KUKA KRL data list: bto.dat

&ACCESS RVP
&REL 2
&PARAM TEMPLATE = C:\KRC\Roboter\Template\vorgabe
&PARAM EDITMASK = *
DEFDAT BTO
;FOLD EXTERNAL DECLARATIONS;%{PE}%V3.2.0,%MKUKATPBASIS,%CEXT,%VCOMMON,%P
;FOLD BAS EXT;%{PE}%V3.2.0,%MKUKATPBASIS,%CEXT,%VEXT,%P
EXT  BAS (BAS_COMMAND  :IN,REAL  :IN )
DECL INT SUCCESS
;ENDFOLD
;FOLD A10 EXT;%{E}%V3.2.0,%MKUKATPARC,%CEXT,%VEXT,%P
EXT  A10 (A_CMD_T  :IN,A_STRT_T  :IN,A_WELD_T  :IN,A_END_T  :IN,INT  :IN )
;ENDFOLD
;FOLD A20 EXT;%{E}%V3.2.0,%MKUKATPA20,%CEXT,%VEXT,%P
EXT  A20 (INT  :IN,WELD_ST  :IN,WELD_FI  :IN,INT  :IN )
;ENDFOLD
;FOLD GRIPPER EXT;%{E}%V3.2.0,%MKUKATPGRIPPER,%CEXT,%VEXT,%P
EXT  H50 (INT  :IN,INT  :IN,INT  :IN,GRP_TYP  :IN )
;ENDFOLD
;FOLD SPOT EXT;%{E}%V3.2.0,%MKUKATPSPOT,%CEXT,%VEXT,%P
EXT  USERSPOT (S_COMMAND  :IN,SPOT_TYPE  :IN )
;ENDFOLD
;FOLD TOUCHSENSE EXT;%{E}%V3.2.0,%MKUKATPTS,%CEXT,%VEXT,%P
EXT  H70 (INT  :IN,SRCH_TYP_2  :OUT,E6POS  :IN,SRCH_TYP_3  :IN,SRCH_TYP_2  :IN,SRCH_TYP_2  :IN,SRCH_TYP_2  :IN,SRCH_TYP_2  :IN,SRCH_TYP_2  :IN,INT  :IN )
;ENDFOLD
;FOLD USER EXT;%{E}%V3.2.0,%MKUKATPUSER,%CEXT,%VEXT,%P
;Make here your modifications
;ENDFOLD
;ENDFOLD

DECL BASIS_SUGG_T LAST_BASIS={POINT1[] "Frente_de_cnc           ",POINT2[] "Frente_de_cnc           ",CP_PARAMS[] "CPDAT1                  ",PTP_PARAMS[] "PDAT1                   ",CONT[] "C_PTP                   ",CP_VEL[] "0.3                     ",PTP_VEL[] "10                      "}
DECL E6POS XFRENTECINTA={x 586.713501,y 475.164886,z 2277.23389,a 88.4521027,b -44.9880409,c -179.531097,s 2,t 43,e1 0.0,e2 0.0,e3 0.0,e4 0.0,e5 0.0,e6 0.0}
DECL FDAT FFrenteCinta={TOOL_NO 0,BASE_NO 0,IPO_FRAME #BASE}
DECL PDAT PPDAT1={VEL 100.0,ACC 100.0,APO_DIST 100.0}
DECL FDAT FFrenteCNC={TOOL_NO 0,BASE_NO 0,IPO_FRAME #BASE}
DECL E6POS XDEJARPINZA2CINTA={x 1620.00403,y -0.00337643898,z 1909.99402,a -110.582497,b 89.9985199,c -110.582397,s 2,t 2,e1 0.0,e2 0.0,e3 0.0,e4 0.0,e5 0.0,e6 0.0}
DECL FDAT FDejarPinza2Cinta={TOOL_NO 2,BASE_NO 0,IPO_FRAME #BASE}
DECL PDAT PPDAT2={VEL 100.0,ACC 100.0,APO_DIST 100.0}
DECL E6POS XDEJARPINZA1CINTA={x -822.804382,y 1453.90796,z 1167.45105,a 3.40687394,b 43.3361893,c -176.740799,s 2,t 35,e1 0.0,e2 0.0,e3 0.0,e4 0.0,e5 0.0,e6 0.0}
DECL FDAT FDejarPinza1Cinta={TOOL_NO 1,BASE_NO 0,IPO_FRAME #BASE}
DECL PDAT PPDAT3={VEL 100.0,ACC 100.0,APO_DIST 100.0}
DECL E6POS XENT1_COGERCINTA={x 444.522186,y 912.39978,z 1228.745,a 87.1254272,b -7.41709614,c -179.732895,s 2,t 43,e1 0.0,e2 0.0,e3 0.0,e4 0.0,e5 0.0,e6 0.0}
DECL FDAT FEnt1_CogerCinta={TOOL_NO 1,BASE_NO 0,IPO_FRAME #BASE}
DECL PDAT PPDAT4={VEL 100.0,ACC 100.0,APO_DIST 100.0}
DECL E6POS XENT2_COGERCINTA={x 175.7229,y 1220.86304,z 1143.29395,a 91.0016403,b -16.5721092,c -179.742203,s 2,t 43,e1 0.0,e2 0.0,e3 0.0,e4 0.0,e5 0.0,e6 0.0}
DECL FDAT FEnt2_CogerCinta={TOOL_NO 1,BASE_NO 0,IPO_FRAME #BASE}
DECL PDAT PPDAT5={VEL 100.0,ACC 100.0,APO_DIST 100.0}
DECL E6POS XENT3COGERCINTA={x 174.258408,y 1264.94495,z 995.101624,a 91.0015488,b -16.5722103,c -179.742203,s 2,t 43,e1 0.0,e2 0.0,e3 0.0,e4 0.0,e5 0.0,e6 0.0}
DECL FDAT FEnt3CogerCinta={TOOL_NO 1,BASE_NO 0,IPO_FRAME #BASE}
DECL PDAT PPDAT6={VEL 100.0,ACC 100.0,APO_DIST 100.0}
DECL LDAT LCPDAT1={VEL 2.0,ACC 100.0,APO_DIST 100.0,APO_FAC 50.0}
DECL E6POS XCOGERCINTA={x 172.789902,y 1308.08704,z 849.818787,a 91.0006485,b -16.5677299,c -179.738998,s 2,t 43,e1 0.0,e2 0.0,e3 0.0,e4 0.0,e5 0.0,e6 0.0}
DECL FDAT FCogerCinta={TOOL_NO 1,BASE_NO 0,IPO_FRAME #BASE}
DECL LDAT LCPDAT2={VEL 2.0,ACC 100.0,APO_DIST 100.0,APO_FAC 50.0}
DECL E6POS XSAL1_COGERCINTA={x 174.258408,y 1264.94495,z 995.101624,a 91.0015488,b -16.5722103,c -179.742203,s 2,t 43,e1 0.0,e2 0.0,e3 0.0,e4 0.0,e5 0.0,e6 0.0}
DECL FDAT FSal1_CogerCinta={TOOL_NO 1,BASE_NO 0,IPO_FRAME #BASE}
DECL LDAT LCPDAT3={VEL 2.0,ACC 100.0,APO_DIST 100.0,APO_FAC 50.0}
DECL E6POS XSAL2_COGERCINTA={x 175.7229,y 1220.86304,z 1143.29395,a 91.0016403,b -16.5721092,c -179.742203,s 2,t 43,e1 0.0,e2 0.0,e3 0.0,e4 0.0,e5 0.0,e6 0.0}
DECL FDAT FSal2_CogerCinta={TOOL_NO 1,BASE_NO 0,IPO_FRAME #BASE}
DECL PDAT PPDAT7={VEL 100.0,ACC 100.0,APO_DIST 100.0}
DECL E6POS XENT1_COGERCNC={x 1664.62,y -787.04303,z 1556.33203,a 3.4404459,b -72.5609131,c 178.200897,s 2,t 42,e1 0.0,e2 0.0,e3 0.0,e4 0.0,e5 0.0,e6 0.0}
DECL FDAT FEnt1_CogerCNC={TOOL_NO 2,BASE_NO 0,IPO_FRAME #BASE}
DECL PDAT PPDAT8={VEL 100.0,ACC 100.0,APO_DIST 100.0}
DECL E6POS XENT2_COGERCNC={x 1791.36096,y -713.231323,z 1242.87,a 2.15886807,b -62.4185295,c 177.698502,s 2,t 42,e1 0.0,e2 0.0,e3 0.0,e4 0.0,e5 0.0,e6 0.0}
DECL FDAT FEnt2_CogerCNC={TOOL_NO 2,BASE_NO 0,IPO_FRAME #BASE}
DECL PDAT PPDAT9={VEL 100.0,ACC 100.0,APO_DIST 100.0}
DECL E6POS XENT3_COGERCNC={x 1968.31201,y -714.600403,z 1150.51599,a 2.13476205,b -62.4179115,c 177.698898,s 2,t 42,e1 0.0,e2 0.0,e3 0.0,e4 0.0,e5 0.0,e6 0.0}
DECL FDAT FEnt3_CogerCNC={TOOL_NO 2,BASE_NO 0,IPO_FRAME #BASE}
DECL LDAT LCPDAT4={VEL 2.0,ACC 100.0,APO_DIST 100.0,APO_FAC 50.0}
DECL E6POS XCOGERCNC={x 2122.44507,y -715.841675,z 1070.07898,a 2.13489294,b -62.4179802,c 177.6987,s 2,t 42,e1 0.0,e2 0.0,e3 0.0,e4 0.0,e5 0.0,e6 0.0}
DECL FDAT FCogerCNC={TOOL_NO 2,BASE_NO 0,IPO_FRAME #BASE}
DECL LDAT LCPDAT5={VEL 2.0,ACC 100.0,APO_DIST 100.0,APO_FAC 50.0}
DECL E6POS XSAL1_COGERCNC={x 2122.44702,y -750.182312,z 1070.07996,a 2.13447905,b -62.4182396,c 177.698898,s 2,t 42,e1 0.0,e2 0.0,e3 0.0,e4 0.0,e5 0.0,e6 0.0}
DECL FDAT FSal1_CogerCNC={TOOL_NO 2,BASE_NO 0,IPO_FRAME #BASE}
DECL LDAT LCPDAT6={VEL 2.0,ACC 100.0,APO_DIST 100.0,APO_FAC 50.0}
DECL E6POS XSAL2_COGERCNC={x 2303.74194,y -787.196472,z 1397.98206,a 2.13354492,b -62.4185104,c 177.699097,s 2,t 42,e1 0.0,e2 0.0,e3 0.0,e4 0.0,e5 0.0,e6 0.0}
DECL FDAT FSal2_CogerCNC={TOOL_NO 2,BASE_NO 0,IPO_FRAME #BASE}
DECL LDAT LCPDAT7={VEL 2.0,ACC 100.0,APO_DIST 100.0,APO_FAC 50.0}
DECL E6POS XENT1_DEJARCNC={x 2008.724,y -885.728271,z 1470.271,a 1.25756299,b -55.0479698,c -179.549301,s 2,t 42,e1 0.0,e2 0.0,e3 0.0,e4 0.0,e5 0.0,e6 0.0}
DECL FDAT FEnt1_DejarCNC={TOOL_NO 1,BASE_NO 0,IPO_FRAME #BASE}
DECL PDAT PPDAT10={VEL 100.0,ACC 100.0,APO_DIST 100.0}
DECL E6POS XENT2_DEJARCNC={x 2273.48389,y -808.585876,z 1205.05798,a 1.25766599,b -55.0479317,c -179.549606,s 2,t 42,e1 0.0,e2 0.0,e3 0.0,e4 0.0,e5 0.0,e6 0.0}
DECL FDAT FEnt2_DejarCNC={TOOL_NO 1,BASE_NO 0,IPO_FRAME #BASE}
DECL PDAT PPDAT11={VEL 100.0,ACC 100.0,APO_DIST 100.0}
DECL E6POS XENT3_DEJARCNC={x 2114.40503,y -752.901978,z 1057.99695,a 1.25682998,b -55.0801506,c -179.549698,s 2,t 42,e1 0.0,e2 0.0,e3 0.0,e4 0.0,e5 0.0,e6 0.0}
DECL FDAT FEnt3_DejarCNC={TOOL_NO 1,BASE_NO 0,IPO_FRAME #BASE}
DECL LDAT LCPDAT8={VEL 2.0,ACC 100.0,APO_DIST 100.0,APO_FAC 50.0}
DECL E6POS XDEJARCNC={x 2113.43701,y -718.692322,z 1058.151,a 1.25690103,b -55.0800896,c -179.556305,s 2,t 42,e1 0.0,e2 0.0,e3 0.0,e4 0.0,e5 0.0,e6 0.0}
DECL FDAT FDejarCNC={TOOL_NO 1,BASE_NO 0,IPO_FRAME #BASE}
DECL LDAT LCPDAT9={VEL 2.0,ACC 100.0,APO_DIST 100.0,APO_FAC 50.0}
DECL E6POS XSAL1_CNC={x 2037.91797,y -721.06012,z 1110.89697,a 1.25862098,b -55.0801697,c -179.557907,s 2,t 42,e1 0.0,e2 0.0,e3 0.0,e4 0.0,e5 0.0,e6 0.0}
DECL FDAT FSal1_CNC={TOOL_NO 1,BASE_NO 0,IPO_FRAME #BASE}
DECL LDAT LCPDAT10={VEL 2.0,ACC 100.0,APO_DIST 100.0,APO_FAC 50.0}
DECL E6POS XSAL2_CNC={x 1572.76794,y -714.070374,z 1503.53406,a 0.854870021,b -43.0494003,c -179.635498,s 2,t 42,e1 0.0,e2 0.0,e3 0.0,e4 0.0,e5 0.0,e6 0.0}
DECL FDAT FSal2_CNC={TOOL_NO 1,BASE_NO 0,IPO_FRAME #BASE}
DECL PDAT PPDAT12={VEL 100.0,ACC 100.0,APO_DIST 100.0}
DECL E6POS XSAL3_CNC={x 1229.31995,y -808.674805,z 1490.52698,a 2.84506607,b -24.9072895,c 179.859299,s 2,t 42,e1 0.0,e2 0.0,e3 0.0,e4 0.0,e5 0.0,e6 0.0}
DECL FDAT FSal3_CNC={TOOL_NO 1,BASE_NO 0,IPO_FRAME #BASE}
DECL PDAT PPDAT13={VEL 100.0,ACC 100.0,APO_DIST 100.0}
DECL PDAT PPDAT14={VEL 100.0,ACC 100.0,APO_DIST 100.0}
DECL E6POS XENT1_DEJARCINTA={x -732.870728,y 1158.88794,z 2270.01904,a 59.0703812,b -89.6684494,c -91.9009628,s 2,t 43,e1 0.0,e2 0.0,e3 0.0,e4 0.0,e5 0.0,e6 0.0}
DECL FDAT FEnt1_DejarCinta={TOOL_NO 2,BASE_NO 0,IPO_FRAME #BASE}
DECL PDAT PPDAT15={VEL 100.0,ACC 100.0,APO_DIST 100.0}
DECL E6POS XENT2_DEJARCINTA={x -1001.48102,y 1524.125,z 1379.88904,a -179.701401,b -42.7616196,c 178.789902,s 2,t 35,e1 0.0,e2 0.0,e3 0.0,e4 0.0,e5 0.0,e6 0.0}
DECL FDAT FEnt2_DejarCinta={TOOL_NO 2,BASE_NO 0,IPO_FRAME #BASE}
DECL PDAT PPDAT16={VEL 100.0,ACC 100.0,APO_DIST 100.0}
DECL E6POS XSAL1_DEJARCINTA={x -732.870728,y 1158.88794,z 2270.01904,a 59.0703812,b -89.6684494,c -91.9009628,s 2,t 43,e1 0.0,e2 0.0,e3 0.0,e4 0.0,e5 0.0,e6 0.0}
DECL FDAT FSal1_DejarCinta={TOOL_NO 2,BASE_NO 0,IPO_FRAME #BASE}
DECL PDAT PPDAT17={VEL 100.0,ACC 100.0,APO_DIST 100.0}
DECL GRP_SUGG_T LAST_GRP={NUMBER[] "2                       ",STATE[] "1                       ",PARAMS[] "GDAT7                   "}
DECL GRP_TYP GGDAT0={G_APO #NO,TIME 0.200000003,CTRL #OFF,DLY 0,DST 1}
DECL GRP_TYP GGDAT2={G_APO #NO,TIME 0.200000003,CTRL #OFF,DLY 0,DST 1}
DECL GRP_TYP GGDAT3={G_APO #NO,TIME 0.200000003,CTRL #OFF,DLY 0,DST 1}
DECL GRP_TYP GCONT={G_APO #YES,TIME 0.0,CTRL #OFF,DLY 0,DST 0}
DECL GRP_TYP GGDAT4={G_APO #NO,TIME 0.200000003,CTRL #OFF,DLY 0,DST 1}
DECL GRP_TYP GGDAT5={G_APO #NO,TIME 0.200000003,CTRL #OFF,DLY 0,DST 1}
DECL GRP_TYP GGDAT6={G_APO #NO,TIME 0.200000003,CTRL #OFF,DLY 0,DST 1}
DECL GRP_TYP GGDAT7={G_APO #NO,TIME 0.200000003,CTRL #OFF,DLY 0,DST 1}
DECL GRP_TYP GCerrar={G_APO #NO,TIME 2.0,CTRL #OFF,DLY 0,DST 1}
DECL GRP_TYP GAbrir={G_APO #NO,TIME 1.0,CTRL #ON,DLY 0,DST 1}
DECL E6POS XSAL3_COJERCNC={x 2103.40088,y -834.78833,z 2002.01294,a 20.8226795,b -87.2193527,c 158.789902,s 2,t 42,e1 0.0,e2 0.0,e3 0.0,e4 0.0,e5 0.0,e6 0.0}
DECL FDAT FSal3_CojerCNC={TOOL_NO 2,BASE_NO 0,IPO_FRAME #BASE}
DECL LDAT LCPDAT11={VEL 2.0,ACC 100.0,APO_DIST 100.0,APO_FAC 50.0}
DECL E6POS XENT1DEJARCINTA={x -732.877625,y 1158.89099,z 2270.01294,a 59.1002197,b -89.6681366,c -91.9304428,s 2,t 43,e1 0.0,e2 0.0,e3 0.0,e4 0.0,e5 0.0,e6 0.0}
DECL FDAT FEnt1DejarCinta={TOOL_NO 2,BASE_NO 0,IPO_FRAME #BASE}
DECL E6POS XDEJARCINTA={x -1001.375,y 1524.11597,z 1154.58203,a 179.620804,b -27.4383392,c -179.7724,s 2,t 35,e1 0.0,e2 0.0,e3 0.0,e4 0.0,e5 0.0,e6 0.0}
DECL FDAT FDejarCinta={TOOL_NO 2,BASE_NO 0,IPO_FRAME #BASE}
DECL E6POS XDejar1Pinza1Cinta={x -186.125397,y 753.741089,z 1449.41602,a 95.8809891,b 44.9203796,c -173.800201,s 2,t 43,e1 0.0,e2 0.0,e3 0.0,e4 0.0,e5 0.0,e6 0.0}
DECL FDAT FDejar1Pinza1Cinta={TOOL_NO 1,BASE_NO 0,IPO_FRAME #BASE}
DECL E6POS XDEJAR11PINZA1CINTA={x 8.99515533,y 1556.49805,z 1254.88403,a -178.753204,b 22.3286991,c -179.640305,s 2,t 43,e1 0.0,e2 0.0,e3 0.0,e4 0.0,e5 0.0,e6 0.0}
DECL FDAT FDejar11Pinza1Cinta={TOOL_NO 1,BASE_NO 0,IPO_FRAME #BASE}
DECL PDAT PPDAT18={VEL 100.0,ACC 100.0,APO_DIST 100.0}
DECL E6POS XDejar12Pinza1Cinta={x -186.133896,y 753.739807,z 1449.41504,a 95.8812408,b 44.9207687,c -173.7995,s 2,t 43,e1 0.0,e2 0.0,e3 0.0,e4 0.0,e5 0.0,e6 0.0}
DECL FDAT FDejar12Pinza1Cinta={TOOL_NO 1,BASE_NO 0,IPO_FRAME #BASE}
DECL E6POS XDEJAR13PINZA1CINTA={x -822.807678,y 1453.89197,z 1331.92896,a 4.23097801,b 54.1295204,c -175.651093,s 2,t 43,e1 0.0,e2 0.0,e3 0.0,e4 0.0,e5 0.0,e6 0.0}
DECL FDAT FDejar13Pinza1Cinta={TOOL_NO 1,BASE_NO 0,IPO_FRAME #BASE}
DECL E6POS XDEJAR14PINZA1CINTA={x -822.157227,y 1482.88794,z 1540.41504,a 46.40839,b 58.6334381,c -133.363007,s 2,t 43,e1 0.0,e2 0.0,e3 0.0,e4 0.0,e5 0.0,e6 0.0}
DECL FDAT FDejar14Pinza1Cinta={TOOL_NO 1,BASE_NO 0,IPO_FRAME #BASE}
DECL PDAT PPDAT19={VEL 100.0,ACC 100.0,APO_DIST 100.0}
DECL FDAT FFrenteaCNC={TOOL_NO 0,BASE_NO 0,IPO_FRAME #BASE}
DECL E6POS XFRENTE_DE_CNC={x 738.229309,y -158.106094,z 2277.23804,a 37.3593597,b -44.987381,c -179.528503,s 2,t 42,e1 0.0,e2 0.0,e3 0.0,e4 0.0,e5 0.0,e6 0.0}
DECL FDAT FFrente_de_cnc={TOOL_NO 0,BASE_NO 0,IPO_FRAME #BASE}
ENDDAT
